KUKA KRL program: clock.src

&ACCESS RVP1
&REL 7
&COMMENT Reset Contador de Pecas
&PARAM TEMPLATE = C:\KRC\Roboter\Template\vorgabe
&PARAM EDITMASK = *
DEF CLOCK( )

; CONTADOR DE PECAS PRODUZIDAS E ZERADO QUANDO ATINGE DEZ HORAS DA NOITE..

IF ($DATE.HOUR == 05) AND ($DATE.MIN == 10) THEN

 I[1] = 0    ; MODELO ACELLO
 I[2] = 0    ; MODELO ACTROS

ENDIF

END
